// TwinCAT 3 PLC project VLSVacuum
// ProgramVersion: 3.1.4023.0
// libraries:
//   L2SI Vacuum Library, * (SLAC)
//   LCLS General, * (SLAC)
//   LCLSVacuumSerialDriverLib, * (SLAC)
//   PMPS, * (SLAC - LCLS)
//   Tc2_SerialCom, * (Beckhoff Automation GmbH)
//   Tc2_Standard, * (Beckhoff Automation GmbH)
//   Tc2_System, * (Beckhoff Automation GmbH)
//   Tc3_Module, * (Beckhoff Automation GmbH)
// project tree:
//   DUTs/ E_STATES.TcDUT (not stored), ST_VRC_NO.TcDUT
//   GVLs/ GVL_COM_VLS.TcGVL (not stored), GVL_PMPS.TcGVL, GVL_VLS.TcGVL
//   / PlcTask.TcTTO (not stored), VLSSerial.TcTTO
//   POUs/ FB_Pfeffier_NoFault_NO.TcPOU, FB_ValveBase_VLS.TcPOU, FB_VGC_VLS.TcPOU, FB_VRC_NO.TcPOU, FB_VRC_NO_FFO_VLS.TcPOU (not stored), MAIN.TcPOU, PRG_PUMP.TcPOU (not stored), PRG_COM.TcPOU (not stored), PRG_VLS_VACUUM.TcPOU, PRG_VLS_WINDOW.TcPOU
// real-time tasks:
//   TASK PlcTask: cycle T#10ms, priority 20, ADS port 350
//   TASK VLSSerial: cycle T#10ms, priority 1, ADS port 351
// I/O:
//   DEVICE Device 1 (EtherCAT), AmsNetId 172.21.132.45.2.1
//     VLS_Term 1 (EK1200)
//     VLS_EP1 (EP2624-0002)
//     VLS_EP2 (EP2338-0001) [EP2338-0001 8 Ch. Dig. Input/Output 24V, 0,5A, M8]
//     VLS_EP3 (EP2339-0021)
//     VLS_EP4 (EP3174-0002) [EP3174-0002 4Ch. Ana. Input +/-10V, 0-10V, 0/4-20mA configurable]
//     VLS_EP5 (EP6002-0002) [EP6002-0002 Interface (RS232/422/485)]
// variable links:
//   VLSVacuum Instance <-> Device 1 (EtherCAT)/VLS_EP1 (EP2624-0002)
//     PlcTask Outputs/GVL_VLS.DS_GCC.q_xHV_DIS <-> Channel 1/Output
//     PlcTask Outputs/GVL_VLS.PTM_01.q_RunDO <-> Channel 3/Output
//   VLSVacuum Instance <-> Device 1 (EtherCAT)/VLS_EP2 (EP2338-0001)
//     PlcTask Inputs/GVL_VLS.PTM_01.i_xAtSpd <-> Channel 1/Input
//     PlcTask Inputs/GVL_VLS.PTM_01.i_xFaultNC <-> Channel 2/Input
//   VLSVacuum Instance <-> Device 1 (EtherCAT)/VLS_EP3 (EP2339-0021)
//     PlcTask Inputs/GVL_VLS.VGC_1.i_xClsLS <-> Channel 7/Input
//     PlcTask Inputs/GVL_VLS.VGC_1.i_xOpnLS <-> Channel 6/Input
//     PlcTask Inputs/GVL_VLS.VGC_W.i_xClsLS <-> Channel 10/Input
//     PlcTask Inputs/GVL_VLS.VGC_W.i_xOpnLS <-> Channel 9/Input
//     PlcTask Outputs/GVL_VLS.VGC_1.q_xOPN_DO <-> Channel 21/Output
//     PlcTask Outputs/GVL_VLS.VGC_W.q_xCLS_DO <-> Channel 24/Output
//   VLSVacuum Instance <-> Device 1 (EtherCAT)/VLS_EP4 (EP3174-0002)
//     PlcTask Inputs/GVL_VLS.DS_GCC.i_iPRESS_R <-> AI Standard Channel 2/Value
//     PlcTask Inputs/GVL_VLS.DS_GPI.i_iPRESS_R <-> AI Standard Channel 1/Value
//     PlcTask Inputs/GVL_VLS.ROUGH_GPI.i_iPRESS_R <-> AI Standard Channel 3/Value
//   VLSVacuum Instance <-> Device 1 (EtherCAT)/VLS_EP5 (EP6002-0002)
//     VLSSerial Inputs/GVL_COM_VLS.stComIn/D[{0..21}] <-> COM TxPDO-Map Inputs Channel 1/Data In {0..21}  (22 links)
//     VLSSerial Inputs/GVL_COM_VLS.stComIn/Status <-> COM TxPDO-Map Inputs Channel 1/Status
//     VLSSerial Outputs/GVL_COM_VLS.stComOut/Ctrl <-> COM RxPDO-Map Outputs Channel 1/Ctrl
//     VLSSerial Outputs/GVL_COM_VLS.stComOut/D[{0..21}] <-> COM RxPDO-Map Outputs Channel 1/Data Out {0..21}  (22 links)

CONFIGURATION VLSVacuum
    RESOURCE PLC ON TwinCAT3
        TASK VLSSerial(INTERVAL := T#10ms, PRIORITY := 1);
        PROGRAM PRG_COM WITH VLSSerial : PRG_COM;
    END_RESOURCE
END_CONFIGURATION

// ---- DUTs/ST_VRC_NO.TcDUT
TYPE ST_VRC_NO EXTENDS ST_ValveBase:
STRUCT
(* Readbacks *)
	//In case VRC is normally open
	{attribute 'pytmc' := '
    pv: CLS_OK;
	field: ONAM CLOSE; 
	field: ZNAM OPEN;
	io: i;
    '}
	xCLS_OK : BOOL := TRUE;
	{attribute 'pytmc' := '
	pv: CLS_SW ;
	field: ONAM CLOSE; 
	field: ZNAM OPEN;
	io: io ;
	'}
	pv_xCLS_SW	: BOOL;
	{attribute 'pytmc' := '
    pv: FORCE_CLS;
	field: ONAM CLOSE; 
	field: ZNAM OPEN;
	io: io;
	'}
	pv_xOvrdCls	:	BOOL;

END_STRUCT
END_TYPE

// ---- GVLs/GVL_PMPS.TcGVL

VAR_GLOBAL

{attribute 'pytmc' := '
    pv: PLC:TST:FF1
    '}
    {attribute 'TcLinkTo' := '.q_xFastFaultOut:=TIIB[PMPS_FFO]^Channel 1^Output'}
    g_FastFaultOutput1  :   FB_HardwareFFOutput;
	
	{attribute 'pytmc' := '
    pv: PLC:TST:FF2
    '}
    {attribute 'TcLinkTo' := '.q_xFastFaultOut:=TIIB[PMPS_FFO]^Channel 2^Output'}
    g_FastFaultOutput2  :   FB_HardwareFFOutput; 
	fbArbiter: FB_Arbiter(1);
	
END_VAR

// ---- GVLs/GVL_VLS.TcGVL
//{attribute 'qualified_only'}
VAR_GLOBAL

	(* OverrideMode *)
	{attribute 'pytmc' := 'pv: VLS:VAC:OVRDON'}
	xSystemOverrideMode_VLS	: BOOL := FALSE; 	

	(* Pfeiffer Turbo Pumps TM700 *)
	{attribute 'TcLinkTo' := 	'.i_xAtSpd			:=	TIIB[VLS_EP2 (EP2338-0001)]^Channel 1^Input;
								 .i_xFaultNC		:=	TIIB[VLS_EP2 (EP2338-0001)]^Channel 2^Input;
								 .q_RunDO			:=	TIIB[VLS_EP1 (EP2624-0002)]^Channel 3^Output;
			 
	'}
	{attribute 'pytmc' := '
		pv: VLS:PTM:01
		io: io
	'}
    PTM_01 : FB_PTM_Pfeiffer;
	PTM_01_xExtIlkOK : Bool;

	// They share the same serial port
	st_Pfeiffer_CTRL 	: ARRAY[1..20] OF ST_PfeifferControl;
	st_Pfeiffer_RBK 	: ARRAY[1..20] OF ST_PfeifferStatus;
	
	fb_PfeifferCom : FB_PFEIFFER_COM;
	
	
	(* Valves *)
	
	{attribute 'pytmc' :=' pv: VLS:VGC:01 '}
	{attribute 'TcLinkTo' := 	'.i_xOpnLS	:=	TIIB[VLS_EP3 (EP2339-0021)]^Channel 6^Input;
								 .i_xClsLS	:=	TIIB[VLS_EP3 (EP2339-0021)]^Channel 7^Input;
								.q_xOPN_DO	:=	TIIB[VLS_EP3 (EP2339-0021)]^Channel 21^Output'}
	VGC_1 : FB_VGC;
	
	{attribute 'pytmc' :=' pv: VLS:VWC:01 '}
	{attribute 'TcLinkTo' := 	'.i_xOpnLS	:=	TIIB[VLS_EP3 (EP2339-0021)]^Channel 9^Input;
								 .i_xClsLS	:=	TIIB[VLS_EP3 (EP2339-0021)]^Channel 10^Input;
								.q_xCLS_DO	:=	TIIB[VLS_EP3 (EP2339-0021)]^Channel 24^Output'}	
	VGC_W : FB_VRC_NO_FFO_VLS; // Is the Window valve NO 
	
	(* Gauges *)
	
	{attribute 'pytmc' :=' pv: VLS:US:GPI '}
	US_GPI	: FB_MKS275;

	{attribute 'pytmc' :=' pv: VLS:US:GCC '}
	US_GCC	: FB_MKS500;

	{attribute 'pytmc' :=' pv: VLS:DS:GPI '}
	{attribute 'TcLinkTo' := 	'.i_iPRESS_R	:=	TIIB[VLS_EP4 (EP3174-0002)]^AI Standard Channel 1^Value		'}
	DS_GPI	: FB_MKS275;

	{attribute 'pytmc' :=' pv: VLS:DS:GCC '}
	{attribute 'TcLinkTo' := 	'.i_iPRESS_R	:=	TIIB[VLS_EP4 (EP3174-0002)]^AI Standard Channel 2^Value;
								 .q_xHV_DIS		:= 	TIIB[VLS_EP1 (EP2624-0002)]^Channel 1^Output	'}		
	DS_GCC	: FB_MKS500;
	
	{attribute 'pytmc' :=' pv: VLS:ROUGH1:GPI '}
	{attribute 'TcLinkTo' := 	'.i_iPRESS_R	:=	TIIB[VLS_EP4 (EP3174-0002)]^AI Standard Channel 3^Value	'}	
	ROUGH_GPI : FB_9XX;
	
	


END_VAR

// ---- POUs/FB_Pfeffier_NoFault_NO.TcPOU
FUNCTION_BLOCK FB_Pfeffier_NoFault_NO EXTENDS FB_Pump
(* This function block does basic controls FOR the Pfeiffer Turbo pump connected to the TM700 and TC400 Controllers.
 Turns off pump in the event of errors/ warnings. Provides interlocking interface.*)

VAR_IN_OUT
	
END_VAR
VAR_INPUT
	i_xExtIlkOK : BOOL; // Connect to external interlock logic, TRUE if not used.
END_VAR
VAR_OUTPUT
	{attribute 'pytmc' := '
    pv: 
	'}
	iq_stPTM : ST_PfeifferPTM;
END_VAR
VAR
	TOF_RESET: TON :=(PT:=T#1S);
	(*IO*)
	i_xAtSpd AT%I*: BOOL; // Normaml operation when true
	i_xFaultNO AT%I*: BOOL; // Error
	i_xWarn AT%I*: BOOL;
 	i_xRemote AT%I*: BOOL;
	
	q_RunDO AT%Q*: BOOL; // Start/Stop for TC110 link this output to the Pumping station bit
	q_PumpingStation AT%Q*: BOOL; // Start/Stop interlock
	q_xRemote AT%Q*: BOOL;
	q_xReset AT%Q*: BOOL;
END_VAR

(* Basic pump supervisory section *)

q_xRemote := TRUE;
(* Interlock Sum *)
iq_stPtm.xExtRunOk:= i_xExtILKOk;
//For compatability with TC110
(*IF iq_stPTM.xExtRunOk THEN
	q_PumpingStation:= TRUE;
ELSE 
	q_PumpingStation:= FALSE;
END_IF*)

IF iq_stPTM.xExtRunOk AND NOT (iq_stPTM.i_xFault) (*OR iq_stPTM.i_xTempFault)*) THEN
	iq_stPTM.q_RunDO:=iq_stPTM.xRunSW;
	q_PumpingStation:=iq_stPTM.xRunSW;
ELSE
	iq_stPTM.xRunSW:=FALSE;
	iq_stPTM.q_RunDO:=FALSE;
	q_PumpingStation:=FALSE;
	//q_xRemote := TRUE;
END_IF


(*Pump STATE*)
IF iq_stPtm.i_xFault THEN 
	iq_stPtm.eState := pumpFAULT;
ELSIF NOT iq_stPtm.q_RunDO AND NOT iq_stPTM.i_xFault THEN
	iq_stPtm.eState := pumpSTOPPED;
ELSIF NOT iq_stPtm.i_xAtSpd  AND iq_stPtm.q_RunDO THEN
	iq_stPtm.eState := pumpSTARTING;
ELSIF iq_stPtm.i_xAtSpd AND iq_stPtm.q_RunDO THEN
	iq_stPtm.eState := pumpRUNNING;
ELSE 
	iq_stPtm.eState := pumpFAULT;
END_IF

(*Error Reset*)
(* to reset the Reset Bit *)
 IF (iq_stPTM.xResetSW ) THEN  
	iq_stPTM.q_xReset := TRUE; 
	q_PumpingStation := TRUE;
 END_IF

 IF (iq_stPTM.xResetSW) AND (iq_stPTM.i_xFault)  THEN  
	q_PumpingStation := TRUE;
 END_IF
 TOF_RESET (IN:= iq_stPTM.q_xReset, Q => );
 IF TOF_RESET.Q THEN 
	iq_stPTM.q_xReset:= FALSE;
	iq_stPTM.xResetSW := FALSE; 
 END_IF

(*Soft IO Mapping*)
ACT_IO();
// Log States and triggers
ACT_Logger();

ACTION ACT_IO:
(*outputs*)
q_RunDO := iq_stPTM.q_RunDO;
q_xReset := iq_stPTM.q_xReset;
//q_xRemote := iq_stPTM.
//q_PumpingStation AT%Q*: BOOL; // Start/Stop
	
(*inputs*)
iq_stPTM.i_xAtSpd:= i_xAtSpd;
iq_stPTM.i_xFault:= i_xFaultNO; 
iq_stPTM.i_xWarn:=  	i_xWarn ;
END_ACTION

ACTION ACT_Logger:
//STATE Logger  
IF NOT i_xExtIlkOK AND ePrevState = pumpRUNNING THEN
 		fbLogger(sMsg:='Lost external interlock while pump was running.', eSevr:=TcEventSeverity.Critical);  	
END_IF


IF ePrevState <> iq_stPTM.eState THEN
	  CASE iq_stPTM.eState OF
		pumpFAULT:
			fbLogger(sMsg:='Pump Fault.', eSevr:=TcEventSeverity.Critical);
  		pumpSTOPPED:
			fbLogger(sMsg:='Pump stopped.', eSevr:=TcEventSeverity.Critical);
		pumpSTARTING:
			fbLogger(sMsg:='Pump starting.', eSevr:=TcEventSeverity.Info);
		pumpRUNNING:
			fbLogger(sMsg:='Pump running.', eSevr:=TcEventSeverity.Info);
	  END_CASE
	  ePrevState := iq_stPTM.eState;  
  END_IF
  
// ILK logger



// Log Action
tAction(CLK:=  iq_stPTM.q_RunDO);
IF tAction.Q THEN fbLogger(sMsg:='Pump commanded to start', eSevr:=TcEventSeverity.Info); END_IF


// Log FAULT
tFault(CLK:= NOT iq_stPTM.i_xFault);
IF tFault.Q THEN fbLogger(sMsg:='Pump Lost Alarm OK bit', eSevr:=TcEventSeverity.Critical); END_IF
END_ACTION

METHOD PUBLIC M_Serial_IO : BOOL
VAR_INPUT
	st_Pfeiffer_RBK: ST_PfeifferStatus;
END_VAR
VAR_IN_OUT
	st_Pfeiffer_CTRL: ST_PfeifferControl;
END_VAR
(* This function block is used to map the IO points from the pfeiffer structures
to the generic turbo structures *)
(*
if (bInit) Then
	bInit := False;
	st_Pfeiffer_CTRL.diSetRotationSpeed_309 := st_Pfeiffer_RBK.diActiveRotationSpeed_309;
END_IF*)

(* Controls *) (* Controls is via DIO*)
st_Pfeiffer_CTRL.xPumpingStation_010 := iq_stPTM.q_RunDO;
//st_Pfeiffer_CTRL.xMotorPump_023 := 1; //Setting always true because parameter 10 alone can enable/disable the pump
//st_Pfeiffer_CTRL.uiPowerPct_708 := iq_stPTM.q_uiPowerPct;
//st_Pfeiffer_CTRL.xErrorAck_009 := iq_stPTM.xResetSW;



(* Readbacks *)
iq_stPTM.i_xAccel := st_Pfeiffer_RBK.xPumpAccelerating_307;
//iq_stPTM.i_xAtSpd := st_Pfeiffer_RBK.xRotationSpeedAttn_306; The Atspd is already linked via Digital I/Os
iq_stPTM.i_diCurSpd := st_Pfeiffer_RBK.diActiveRotationSpeed_309;
iq_stPTM.i_diPwr := st_Pfeiffer_RBK.diDrivePower_316;
iq_stPTM.i_diElecTemp := st_Pfeiffer_RBK.diTempElec_326;
iq_stPTM.i_diBtmTemp := st_Pfeiffer_RBK.diTempPmpBot_330;
iq_stPTM.i_diBrngTemp := st_Pfeiffer_RBK.diTempBearng_342;
iq_stPTM.i_diMtrTemp := st_Pfeiffer_RBK.diTempMotor_346;
iq_stPTM.i_uiPowerPctRbk := st_Pfeiffer_RBK.uiPowerPct_708;
iq_stPTM.i_rCurrentMon :=  st_Pfeiffer_RBK.lrDriveCurrent_310;
iq_stPTM.xCommTimeout	:=	st_Pfeiffer_RBK.xTimeout;
iq_stPTM.i_iErrorCode := st_Pfeiffer_RBK.iErrorCode_303;
iq_stPTM.i_iWarningCode := st_Pfeiffer_RBK.iWarningCode_303;

(* Check that error acknowledgment is processed *)
IF st_Pfeiffer_RBK.xErrorAcknowledged THEN
	st_Pfeiffer_RBK.xErrorAcknowledged := FALSE;
	st_Pfeiffer_CTRL.xErrorAck_009 := FALSE;
	iq_stPTM.xResetSW := FALSE;
END_IF

IF st_Pfeiffer_RBK.sErrorCode_303 = '' THEN
	;
ELSIF st_Pfeiffer_RBK.sErrorCode_303 <> '000000' THEN
iq_stPTM.i_xFault := TRUE;
ELSE
iq_stPTM.i_xFault := FALSE;
END_IF

iq_stPTM.i_dSetSpd := LIMIT (0, iq_stPTM.i_dSetSpd, 1500); // 1500 nominal frequency
IF ( iq_stPTM.i_dSetSpd <>0) THEN
	st_Pfeiffer_CTRL.iSetRotationSpeed_707 := DINT_TO_INT(iq_stPTM.i_dSetSpd * 100/1500);
	st_Pfeiffer_CTRL.iSetRotationSpeed_707 := LIMIT(20, st_Pfeiffer_CTRL.iSetRotationSpeed_707 ,100); // Manual Page 18
END_IF
END_METHOD

END_FUNCTION_BLOCK

// ---- POUs/FB_ValveBase_VLS.TcPOU
FUNCTION_BLOCK FB_ValveBase_VLS
VAR_INPUT
END_VAR
VAR_OUTPUT
END_VAR
VAR
	// For logging
    fbLogger : FB_LogMessage := (eSubsystem:=E_SubSystem.VACUUM);
   // ePrevState : E_ValvePositionState;
    tErrorPresent : R_TRIG;
    tAction : R_TRIG; // Primary action of this device (OPN_DO, etc.)
    tOverrideActivated : R_TRIG;
END_VAR

ACTION ACT_Logger:

END_ACTION

END_FUNCTION_BLOCK

// ---- POUs/FB_VGC_VLS.TcPOU
(* This function block implements basic functionality for Isolation Gate Valves*)
(* This function block interlock is as follows:
1. The valve can be opened when the difference between the pressures on both sides is
less than the maximum differential pressure.
2. This rule persists until the pressures on both sides are lower than the vacuum-setpoint.
3. Once at-vac, the valve will close if the pressure on either side rises above the setpoint.*)
(*This function block also implements PMPS and EPS interlocks, as well as Fast MPS trigger*)
FUNCTION_BLOCK FB_VGC_VLS Extends FB_ValveBase
VAR_IN_OUT
END_VAR
VAR_INPUT
	(*Upstream Gauge, usually ion gauge*)
	i_stUSG	:	ST_VG;
	(*Downstream Gauge, usually ion gauge*)
	i_stDSG	:	ST_VG;
	{attribute 'pytmc' := '
    pv: Dis_DPIlk
	'}
	i_xDis_DPIlk : BOOL := FALSE;  (* Set to true when calling the function to disable the differential pressure interlock *)
	{attribute 'pytmc' := '
    pv: EPS_OPN_OK
	'}
	i_xEPS_OPN_OK:	BOOL	:= TRUE; (*External EPS interlock, Set to TRUE when no EPS interlock is required, otherwise set to correct interlock signal*)
	{attribute 'pytmc' := '
    pv: EPS_CLS_OK
	'}
	i_xEPS_CLS_OK:	BOOL	:= TRUE; (*External EPS interlock, Set to TRUE when no EPS interlock is required, otherwise set to correct interlock signal*)
	
	{attribute 'pytmc' := '
    pv: MPS_OK
	'}
	i_xPMPS_OK:	BOOL	; (*External MPS interlock, Set to TRUE when no PMPS interlock is required*)
	i_xExt_OK: BOOL; (*Other External Interlock, Set to True when no external interlock is required. If this Valve is neigboring a Fast Shutter this should be linked to the fast shutter xVAC_FAULT_OK*)
	i_xOverrideMode : BOOL; (*To be linked to global override bit. This Overrides Vacuum logic only, EPS, MPS and PMPS are still enforces*)
	// Reset fault
	{attribute 'pytmc' := '
    pv: FF_Reset
	'}
    i_xReset: BOOL;
END_VAR
VAR_OUTPUT
	{attribute 'pytmc' := '
    pv:
	'}
	iq_stValve : ST_VGC; (* All valve data and states will be in this struct*)
	
END_VAR

VAR
	{attribute 'instance-path'}
	{attribute 'noinit'}
	sPath: STRING;
	rDiffPressAllowed	:	REAL := 22.5; // Torr, Default value comes from Vat Valve Manual
	rDiffPress : REAL;
	set : BOOL;
    reset: BOOL;
	  
	xFirstPass	:	BOOL;
	fbFSInit		:	R_TRIG;
	
	tonDelOK : TON;
	rtOK	:	R_TRIG;
	tonOvrd	:	TON;
	rtOpen	:	R_TRIG;
	ftClose: F_TRIG;
	
	tDelOK	:	TIME := T#60S;
	tOvrd	:	TIME := T#10s;
	ePrevState : E_VGC;
	
	(* Timeouts*)
	tTimeOutDuration: TIME:= T#10S;
	tOPNtimeout: TON;
	tCLStimeout:TON;
	
	
	
	(*IO*)
	i_xOpnLS	AT%I*: BOOL;
	i_xClsLS	AT%I*: BOOL;
	q_xOPN_DO	AT%Q*: BOOL;
    
  
END_VAR

(* Vacuum gate valve
A. Wallace
16-10-29

A gate valve isolates vacuum volumes. Ideally it can be opened when a system is vented
to allow for faster pumping, and will close when high vacuum is lost.

The following behavior is good for valves in something like a gas attenuator.
This function block does the following:
1. The valve can be opened when the difference between the pressures on both sides is
less than the maximum differential pressure.
2. This rule persists until the pressures on both sides are lower than the vacuum-setpoint.
3. Once at-vac, the valve will close if the pressure on either side rises above the setpoint.

Alternatively, the differential pressure interlock can be disabled so the valve may only be opened
if the pressure on both sides is lower than the at-vacuum-setpoint. You want this behavior if 
the valve is to be used in a UHV section.

Hysteresis is employed to ensure a smooth transition from vented/pumping down, to at-vac.

Finally, an override system is built in so you can bypass all the interlocking logic and 
get back online.
*)
(* 10/1/2018 Margaret Ghaly included EPS, PMPS Checkes and MPS trigger signals*)

ACT_Init();
(*IO Mapping*)
ACT_IO();
A_Override();
A_PositionCheck();
ACT_ResetAlarms();
A_EPS();
// Main logic the very last call right before IO
ACT_Main();
(*IO Mapping*)
ACT_IO();
A_Logger();

ACTION A_EPS:
ftClose(CLK:= iq_stValve.pv_xOPN_SW);
rtOpen(CLK:= iq_stValve.pv_xOPN_SW);


(* If Epics Command to close the Valve, check if PMPS and EPS are ok, otherwise Keep command set to open valve *)
// Check a falling edge on the open switch, which means that the valve is commanded to close
IF (ftClose.Q) THEN
	// check that the valve is allowed to close, and that it was already in the open position otherwise, he command is to be ingonred and reset
	IF NOT(i_xEPS_CLS_OK) AND (iq_stValve.q_xOPN_DO) THEN iq_stValve.pv_xOPN_SW := TRUE; END_IF;
END_IF

// if switch pv has been switched to open
IF (rtOpen.Q) THEN 
	// if the EPS interlock the valve from openening, the switch pv is reset to false i.e ignoring the action
	IF NOT (i_xEPS_OPN_OK) THEN  iq_stValve.pv_xOPN_SW := FALSE; END_IF
END_IF
END_ACTION

ACTION A_Logger:
// Log valve timeouts
tErrorPresent(CLK:=iq_stValve.bErrorPresent);
IF tErrorPresent.Q THEN fbLogger(sMsg:=iq_stValve.sErrorMessage, eSevr:=TcEventSeverity.Warning); END_IF

// Log valve open
tAction(CLK:= iq_stValve.q_xOPN_DO);
IF tAction.Q THEN fbLogger(sMsg:='Valve commanded open', eSevr:=TcEventSeverity.Info); END_IF

// Log override mode enabled
tOverrideActivated(CLK:= (tonOvrd.Q AND i_xOverrideMode));
IF tOverrideActivated.Q THEN fbLogger(sMsg:='Valve override mode activated', eSevr:=TcEventSeverity.Warning); END_IF
END_ACTION

ACTION A_Override:
(* Override logic *)
(* Goal: give ability to override, but do so in a way that people won't forget it.
Solution: Override only after ten seconds of override, protect against blips,
when the valve permission goes true for more than ten seconds consistently, remove override
*)

tonDelOK(IN:=iq_stValve.xOPN_OK, PT:=tDelOK);
rtOK(CLK:=tonDelOK.Q);
IF rtOK.Q AND iq_stValve.pv_xOvrdOpn THEN 
	if (iq_stValve.eState = OPEN) AND (i_xOverrideMode) AND (iq_stValve.pv_xOvrdOpn) THEN iq_stValve.pv_xOPN_SW := TRUE; END_IF //for seamless transition   
   	iq_stValve.pv_xOvrdOpn :=FALSE; // reset the overrride open bit
	//Log
    fbLogger(sMsg:='Override expired', eSevr:=TcEventSeverity.Warning);
    
END_IF

//Override timer
tonOvrd(IN:=iq_stValve.pv_xOvrdOpn, PT:=tOvrd);
END_ACTION

ACTION A_PositionCheck:


///Check valve position
IF iq_stValve.i_xClsLS AND  iq_stValve.i_xOpnLS THEN
	iq_stValve.eState:=INVALID;
ELSIF NOT iq_stValve.i_xClsLS AND iq_stValve.i_xOpnLS AND iq_stValve.q_xOPN_DO THEN 
	iq_stValve.eState:=OPEN;
ELSIF iq_stValve.i_xClsLS AND NOT iq_stValve.i_xOpnLS AND NOT iq_stValve.q_xOPN_DO THEN 
	iq_stValve.eState:=CLOSED;
ELSIF NOT iq_stValve.i_xClsLS AND NOT iq_stValve.i_xOpnLS THEN 
	iq_stValve.eState:=MOVING;
ELSE
	iq_stValve.eState:=INVALID;
END_IF


///Check valve moving postion timout
IF NOT iq_stValve.i_xClsLS AND tCLStimeout.Q THEN 
	iq_stValve.bErrorPresent := TRUE;
	iq_stValve.sErrorMessage := ' Close Timeout';
ELSIF NOT iq_stValve.i_xOpnLS AND tOPNtimeout.Q THEN 
	iq_stValve.bErrorPresent := TRUE; 
	iq_stValve.sErrorMessage := ' Open Timeout';
END_IF
IF (iq_stValve.eState=INVALID) THEN
	iq_stValve.bErrorPresent := TRUE; 
	iq_stValve.sErrorMessage := CONCAT(sPath,' Invalid Valve Position');
END_IF


(*Timers*)
tOPNtimeout(IN:= iq_stValve.q_xOPN_DO, PT := tTimeOutDuration );
tCLStimeout(IN:= NOT iq_stValve.q_xOPN_DO, PT := tTimeOutDuration);
END_ACTION

ACTION ACT_Init:
fbFSInit( CLK := TRUE, Q => xFirstPass);
(* On first PLC pass, put valve into vented state, which implies a closed valve *)
IF xFirstPass THEN
	iq_stValve.eVGC_State := Vented;
	iq_stValve.pv_xOPN_SW := FALSE;
END_IF
END_ACTION

ACTION ACT_IO:
(*inputs*)
iq_stValve.i_xOpnLS := 	i_xOpnLS;
iq_stValve.i_xClsLS:=	i_xClsLS;
iq_stValve.xEXT_OK := i_xEXT_OK;
iq_stValve.xOverrideMode := i_xOverrideMode;
(*outputs*)
q_xOPN_DO:= iq_stValve.q_xOPN_DO;
END_ACTION

ACTION ACT_Main:

// Update hysteresis
///////////////////////////////////////////////////
IF iq_stValve.rAT_VAC_SP_LAST <> iq_stValve.rAT_VAC_SP OR xFirstPass THEN
	iq_stValve.rAT_VAC_SP_LAST := iq_stValve.rAT_VAC_SP;
	iq_stValve.rAT_VAC_HYS := iq_stValve.rHYST_PERC * iq_stValve.rAT_VAC_SP;
END_IF

iq_stValve.rAT_VAC_HYS := LIMIT(0, iq_stValve.rAT_VAC_HYS, iq_stValve.rAT_VAC_SP);
IF iq_stValve.rAT_VAC_SP <> 0 THEN
	IF iq_stValve.rHYST_PERC <> (iq_stValve.rAT_VAC_HYS / iq_stValve.rAT_VAC_SP) THEN
		iq_stValve.rHYST_PERC := LIMIT(0, (iq_stValve.rAT_VAC_HYS / iq_stValve.rAT_VAC_SP) ,1);
	END_IF
END_IF
// Valve at vacuum check
///////////////////////////////////////////////////
	set := i_stUSG.rPRESS < iq_stValve.rAT_VAC_HYS AND i_stDSG.rPRESS < iq_stValve.rAT_VAC_HYS AND i_stUSG.xPRESS_OK AND i_stDSG.xPRESS_OK;
 	iq_stValve.xAT_VAC S= set;
	reset := i_stUSG.rPRESS > iq_stValve.rAT_VAC_SP OR i_stDSG.rPRESS > iq_stValve.rAT_VAC_SP OR NOT i_stUSG.xPRESS_OK OR NOT i_stDSG.xPRESS_OK;
	iq_stValve.xAT_VAC R= reset;
	
// Differential pressure check
///////////////////////////////////////////////////
	(* Calc the differential pressure across the valve *)
	rDiffPress := ABS(i_stUSG.rPRESS - i_stDSG.rPRESS);
	
	(* As long as the differential pressure is less than 30mbar, the valve is allowed to open *)
	IF rDiffPress <= rDiffPressAllowed AND i_stUSG.xPRESS_OK AND i_stDSG.xPRESS_OK THEN
		iq_stValve.xDP_OK := TRUE;
	ELSE
		iq_stValve.xDP_OK	:= FALSE;
		(* If the differential pressure is exceeded, even when the valve is open,
		the state is unexpected and triggers a fault, because it suggests that something
		is wrong with the valve, or gauges or mapping or there is a major leak on one side.*)
		iq_stValve.eVGC_State := ERR_DiffPress;
        iq_stValve.xERR_DifPres := TRUE;
	END_IF

// Valve state
///////////////////////////////////////////////////
CASE iq_stValve.eVGC_State OF
	Vented: (* The Vented state is used during pump down *)
        //Log new state
        IF ePrevState <> iq_stValve.eVGC_State THEN
            fbLogger(sMsg:='Vented', eSevr:=TcEventSeverity.Info);
            ePrevState := iq_stValve.eVGC_State;
		END_IF
        
		(* Assuming the pump down went well, we are now at vacuum on both sides,
		so we move to the vacuum state, otherwise remain in the vented state *)
		IF iq_stValve.xAT_VAC AND (NOT (iq_stValve.xERR_DifPres)) AND NOT (NOT (iq_stValve.xERR_SP)) and NOT (NOT (iq_stValve.xERR_ExtFault))THEN
		    iq_stValve.eVGC_State := AtVacuum;
		ELSE
		    iq_stValve.eVGC_State := Vented;
		END_IF
	
	AtVacuum:
        //Log new state
        IF ePrevState <> iq_stValve.eVGC_State THEN
            fbLogger(sMsg:='Vacuum setpoint satisfied', eSevr:=TcEventSeverity.Info);
            ePrevState := iq_stValve.eVGC_State;
		END_IF
        
		IF iq_stValve.xAT_VAC THEN
		(* If both pressure setpoints are made,
		then enable the differential pressure interlock, regardless of the valve state
		assuming we're using some kind of ion gauge where a pressure setpoint cannot be higher than 1E-4 T *)
		iq_stValve.eVGC_State := AtVacuum;
				
		ELSE
		
			(* If the valve is open (or in an unknown state) and either gauge is not at it's vacuum setpoint,
			we have a loss of vacuum error *)
			IF (iq_stValve.i_xOpnLS OR (NOT iq_stValve.i_xOpnLS AND NOT iq_stValve.i_xClsLS)) THEN
				iq_stValve.eVGC_State := ERR_LostVac;
				iq_stValve.xERR_SP := TRUE; //TAW changed this to the ERR_SP bool because I think that's what it was intended to be?
		
			(* Alternatively, if the valve is already closed and we lose pressure on one side,
			it was probably intentional venting, so we calmly move back to venting mode, and
			disable the differential pressure interlock *) //?? 
			ELSIF iq_stValve.i_xClsLS THEN
				iq_stValve.eVGC_State := Vented;
			END_IF
		
		END_IF
	
	ERR_DiffPress:
        //Log new state
        IF ePrevState <> iq_stValve.eVGC_State THEN
            fbLogger(sMsg:='Potential accidental vent.', eSevr:=TcEventSeverity.Critical);
            ePrevState := iq_stValve.eVGC_State;
		END_IF
        
		IF NOT (iq_stValve.xERR_DifPres) THEN
			iq_stValve.eVGC_State := Vented;
		END_IF
		
	
	ERR_LostVac:
        //Log new state
        IF ePrevState <> iq_stValve.eVGC_State THEN
            fbLogger(sMsg:='Unexpected loss of vacuum while valve was open.', eSevr:=TcEventSeverity.Critical);
            ePrevState := iq_stValve.eVGC_State;
		END_IF
		IF NOT (iq_stValve.xERR_SP) THEN
			iq_stValve.eVGC_State := Vented;
		END_IF
		
	ERR_ExtFault:
        //Log new state
        IF ePrevState <> iq_stValve.eVGC_State THEN
            fbLogger(sMsg:='Lost external interlock while valve was open.', eSevr:=TcEventSeverity.Critical);
            ePrevState := iq_stValve.eVGC_State;
		END_IF
		IF NOT (iq_stValve.xERR_ExtFault) AND (NOT i_xExt_OK) THEN
			iq_stValve.eVGC_State := Vented;
		END_IF
END_CASE

IF (NOT i_xExt_OK) THEN
	iq_stValve.eVGC_State := ERR_ExtFault;
	iq_stValve.xERR_ExtFault := TRUE;
END_IF

// Interlock evaluation - with bypass for DP ILK bypass
///////////////////////////////////////////////
IF i_xDis_DPIlk THEN
	iq_stValve.xOPN_OK := iq_stValve.xEXT_OK; // AND iq_stValve.xDP_OK ;
ELSE
	iq_stValve.xOPN_OK := iq_stValve.xEXT_OK AND iq_stValve.xAT_VAC;
END_IF

(* Valve operation *)
if NOT (iq_stValve.xOPN_OK) THEN iq_stValve.pv_xOPN_SW:= FALSE; END_IF // redundant??
(* Here's where the valve opens *)
iq_stValve.q_xOPN_DO := (iq_stValve.pv_xOPN_SW AND iq_stValve.xOPN_OK) OR (tonOvrd.Q AND i_xOverrideMode);
END_ACTION

ACTION ACT_ResetAlarms:
iq_stValve.xERR_DifPres R= iq_stValve.pv_xAlmRst;
iq_stValve.xERR_SP R= iq_stValve.pv_xAlmRst;
iq_stValve.bErrorPresent R= iq_stValve.pv_xAlmRst;

IF ( iq_stValve.pv_xAlmRst) THEN
	iq_stValve.sErrorMessage :='';
END_IF
END_ACTION

METHOD PUBLIC M_IsClosed : BOOL
VAR_INPUT
END_VAR
M_IsClosed := (This^.iq_stValve.eState = E_ValvePositionState.CLOSED);
END_METHOD

METHOD PUBLIC M_IsOpen : BOOL
VAR_INPUT
END_VAR
M_IsOpen := (This^.iq_stValve.eState = E_ValvePositionState.OPEN);
END_METHOD

// Use this Methode to Open or close the valve by setting the OPN_SW to the input value.
METHOD PUBLIC M_Set_OPN_SW : BOOL
VAR_INPUT
		value:BOOL;
END_VAR
This^.iq_stValve.pv_xOPN_SW := value;
END_METHOD

END_FUNCTION_BLOCK

// ---- POUs/FB_VRC_NO.TcPOU
(* This function block is different from the regular VRC in that CLOSING must be permitted. *)
FUNCTION_BLOCK FB_VRC_NO EXTENDS FB_Valve
VAR_IN_OUT

END_VAR
VAR_INPUT

	i_xExtILK_OK : BOOL; //Connect to Interlock logic condition(e.g F_TURBO_VRC_ILK Function), otherwise, Set to True if the valve is not interlocked
	i_xOverrideMode : BOOL; (*To be linked to global override bit. This Overrides Vacuum logic only, EPS, MPS and PMPS are still enforces*)

END_VAR
VAR_OUTPUT
	{attribute 'pytmc' := '
    pv:
	'}
		iq_stValve : ST_VRC_NO;
END_VAR
VAR

	{attribute 'noinit'}
	sPath: STRING;
	xFirstPass	:	BOOL;
	fbFSInit		:	R_TRIG;
	tonOvrd	:	TON;
	tonDelOK : TON;
	rtOK	:	R_TRIG;
	tOvrd	:	TIME := T#10s;
	(* Timeouts*)
	tTimeOutDuration: TIME:= T#30S;
	tOPNtimeout: TON;
	tCLStimeout:TON;
	

(*IO*)
	i_xOpnLS	AT%I*: BOOL;
	i_xClsLS	AT%I*: BOOL;
	q_xCLS_DO	AT%Q*: BOOL;

END_VAR

(* This function block is different from the regular VRC in that CLOSING must be permitted. *)

(* On first PLC pass, put valve into vented state, which implies a closed valve *)
fbFSInit( CLK := TRUE, Q => xFirstPass);
IF xFirstPass THEN
	iq_stValve.pv_xCLS_SW := FALSE;
END_IF




///Check valve position
IF iq_stValve.i_xClsLS AND  iq_stValve.i_xOpnLS THEN
	iq_stValve.eState:=INVALID;
ELSIF NOT iq_stValve.i_xClsLS AND iq_stValve.i_xOpnLS AND iq_stValve.q_xOPN_DO THEN 
	iq_stValve.eState:=OPEN;
ELSIF iq_stValve.i_xClsLS AND NOT iq_stValve.i_xOpnLS AND NOT iq_stValve.q_xOPN_DO THEN 
	iq_stValve.eState:=CLOSED;
ELSIF NOT iq_stValve.i_xClsLS AND NOT iq_stValve.i_xOpnLS THEN 
	iq_stValve.eState:=MOVING;
ELSE
	iq_stValve.eState:=INVALID;
END_IF


(*evaluate Valve CLose external interlock*)
iq_stValve.xCLS_OK := i_xExtILK_OK;
IF NOT iq_stValve.xCLS_OK and NOT tonOvrd.Q THEN
	iq_stValve.pv_xCLS_SW := FALSE;
END_IF


(* Override logic *)
(* Goal: give ability to override, but do so in a way that people won't forget it.
Solution: Override only after ten seconds of override, protect against blips,
when the valve permission goes true for more than ten seconds consistently, remove override
*)

tonDelOK(IN:=iq_stValve.xCLS_OK, PT:=T#10S);
rtOK(CLK:=tonDelOK.Q);
IF rtOK.Q AND iq_stValve.pv_xOvrdCls THEN 
	iq_stValve.pv_xOvrdCls :=FALSE; 
	if (iq_stValve.eState=CLOSED) AND (i_xOverrideMode) THEN iq_stValve.pv_xCLS_SW := TRUE; END_IF
    //Log
    fbLogger(sMsg:='Override expired', eSevr:=TcEventSeverity.Warning);
END_IF

//Override timer
tonOvrd(IN:=iq_stValve.pv_xOvrdCls, PT:=tOvrd);

(* Here's where the valve Actuates *)
q_xCLS_DO := ((iq_stValve.xCLS_OK  AND iq_stValve.pv_xCLS_SW)OR (tonOvrd.Q AND i_xOverrideMode));
iq_stValve.q_xOPN_DO := NOT q_xCLS_DO;



///Check valve moving position timout
IF NOT iq_stValve.i_xClsLS AND tCLStimeout.Q THEN 
	iq_stValve.bErrorPresent := TRUE;
	//iq_stValve.sErrorMessage := ' Close Timeout';
ELSIF NOT iq_stValve.i_xOpnLS AND tOPNtimeout.Q THEN 
	iq_stValve.bErrorPresent := TRUE; 
	//iq_stValve.sErrorMessage := ' Open Timeout';
END_IF
IF (iq_stValve.eState=INVALID) THEN
	iq_stValve.bErrorPresent := TRUE; 
	//iq_stValve.sErrorMessage := CONCAT(sPath,' Invalid Valve Position');
END_IF

(*Timers*)
tOPNtimeout(IN:= iq_stValve.q_xOPN_DO, PT := tTimeOutDuration );
tCLStimeout(IN:= NOT iq_stValve.q_xOPN_DO, PT := tTimeOutDuration);


(*Soft IO Mapping*)
ACT_IO();

// Log States and triggers
ACT_Logger();

ACTION ACT_IO:
(*inputs*)
iq_stValve.i_xOpnLS := 	i_xOpnLS;
iq_stValve.i_xClsLS:=	i_xClsLS;
//iq_stValve. := i_xEXT_OK;
iq_stValve.xOverrideMode := i_xOverrideMode;
(*outputs*)
//q_xOPN_DO:= iq_stValve.q_xOPN_DO;
END_ACTION

METHOD M_IsClosed : BOOL
VAR_INPUT
END_VAR
M_IsClosed := (This^.iq_stValve.eState = E_ValvePositionState.CLOSED);
END_METHOD

METHOD M_IsOpen : BOOL
VAR_INPUT
END_VAR
M_IsOpen := (This^.iq_stValve.eState = E_ValvePositionState.OPEN);
END_METHOD

METHOD M_Set_CLS_W : BOOL
VAR_INPUT
	value:BOOL;
END_VAR
This^.iq_stValve.pv_xCLS_SW := value;
END_METHOD

END_FUNCTION_BLOCK

// ---- POUs/MAIN.TcPOU
PROGRAM MAIN
VAR
	// Variable for VLS upstream pressure bit
	{attribute 'pytmc' := '
	pv: EXT_PRESS_OK ;
	field: ZNAM NOT OK ;
	field: ONAM OK ;
	io: i ;
	'}
	bVLS_Press_OK : BOOL := FALSE; // TRUE : OK to open gate valve, FALSE : not OK to open gate valve
	
//	stPTM : ST_PfeifferControl;
//	fbPTM : FB_PTM_Pfeiffer;
END_VAR

(* Example main program to show how to incorporate the VLS vacuum program *)

PRG_VLS_VACUUM();

END_PROGRAM

// ---- POUs/PRG_VLS_VACUUM.TcPOU
PROGRAM PRG_VLS_VACUUM
VAR


END_VAR
VAR_INPUT
	bVLS_Ext_Press : BOOL := FALSE; // external interlock bit for window control
END_VAR

// VLS Vacuum Logic
PRG_VLS_WINDOW(bExtPress := bVLS_Ext_Press); // run the vacuum program with interlock bit

// VLS Pump
PRG_PUMP();

END_PROGRAM

// ---- POUs/PRG_VLS_WINDOW.TcPOU
PROGRAM PRG_VLS_WINDOW
VAR
	xFirstPass		: BOOL;
	fbFSInit		: R_TRIG;
	
	state			: E_STATES;

	bOverride		: BOOL;
	bSetup			: BOOL;
	

END_VAR
VAR_INPUT
	bExtPress		: BOOL := FALSE; // Input for external interlock with hutch vacuum system
END_VAR

fbFSInit( CLK := TRUE, Q => xFirstPass);
(* On first PLC pass, put valve into init state*)
IF xFirstPass THEN
	state:= E_STATES.INIT;
	bOverride := FALSE;
	bSetup := FALSE;
END_IF


//STATE ACTIONS
CASE state OF

 E_STATES.INIT: 
		VGC_1.M_Set_OPN_SW(FALSE); //Isolation Valve closed
		VGC_W.M_Set_CLS_SW(FALSE); // Window valve OPEN
		VGC_1.i_xOverrideMode := VGC_W.i_xOverrideMode := FALSE;
		//Transition
		if (VGC_1.M_IsClosed() AND VGC_W.M_IsOpen()) THEN
			state:= E_STATES.NOT_SAFE;
		END_IF
		
E_STATES.NOT_SAFE: // System is not allowed to actuate, i.e all interlocks are in effect
	VGC_1.M_Set_OPN_SW(VGC_1.iq_stValve.q_xOPN_DO );
 	//C_1.i_xExt_OK := VGC_1.i_xEPS_OPN_OK := VGC_1.i_xEPS_CLS_OK:= FALSE; 
	VGC_W.i_xExtILK_OK:= FALSE; 
	VGC_1.i_xOverrideMode := VGC_W.i_xOverrideMode := FALSE;

	//Transition
	//IF (US_GCC.IG.xAT_VAC AND DS_GCC.IG.xAT_VAC) THEN state:= E_STATES.READY; END_IF
	IF (bExtPress AND DS_GCC.IG.xAT_VAC) THEN state:= E_STATES.READY; END_IF
	
	
	
 E_STATES.READY: // OK to MOVE
 	// Release the external interlock so the differential pressure inlk is in effect
 	VGC_1.i_xExt_OK:= VGC_1.i_xEPS_OK :=TRUE;
	//permission to insert window valve only when US vacuum is good??
	VGC_W.i_xExtILK_OK:= bExtPress;
	// Valves  alternate positions.
	If (VGC_W.M_IsClosed()) THEN  VGC_1.M_Set_OPN_SW(TRUE);
	ELSIF (VGC_W.M_IsOpen()) THEN VGC_1.M_Set_OPN_SW(FALSE);
	END_IF
	
 
 E_STATES.OVERRIDE: 
	// Override Mode is enabled for all valves
 	VGC_1.i_xOverrideMode :=VGC_W.i_xOverrideMode := TRUE;
	// Exit of Override mode always goes back to init
 	IF NOT(bOverride) THEN state:= E_STATES.INIT; END_IF
	
	
 E_STATES.SETUP: 
	// Window valve remains retracted
 	VGC_W.i_xExtILK_OK := FALSE; 
	// Isolation valves operates like standard gate valves 
	VGC_1.i_xExt_OK := TRUE;
	// exit to init just to be safe?
	IF NOT(bSetup) THEN state:= E_STATES.INIT; END_IF
END_CASE


// STATE TRANSITIONS
// the system can go to setup state from any other state except override
IF (bSetup) AND (state<>E_STATES.OVERRIDE) THEN state:= E_STATES.SETUP; 
// the system can go to override state from any other state except setup
ELSIF (bOverride) AND (state<>E_STATES.SETUP) THEN state:= E_STATES.OVERRIDE;
//Loss of at vac signal makes the system go to init/not safe to move state
ELSIF (NOT bExtPress) OR (NOT DS_GCC.IG.xAT_VAC) THEN state:= E_STATES.INIT;
//ELSIF (NOT US_GCC.IG.xAT_VAC) OR (NOT DS_GCC.IG.xAT_VAC) THEN state:= E_STATES.INIT;
END_IF 


// Instantiate function blocks
US_GPI(PG=>);
//US_GCC(PG:=US_GPI.PG);
DS_GPI(PG=>);
DS_GCC(PG:=DS_GPI.PG , IG=> , bEP := TRUE );

ROUGH_GPI.M_SetBits(32767);
ROUGH_GPI(PG=>);

VGC_1(
	i_stUSG:= US_GCC.IG , 
	i_stDSG:= DS_GCC.IG , 
	i_xDis_DPIlk:= FALSE , 
	i_xPMPS_OK:= , 
	i_xEPS_OK:= , 
	i_xExt_OK:= , 
	i_xOverrideMode:= , 
	i_xReset:= , 
	i_xIsAperture:= FALSE, 
	i_sDevName:= , 
	i_nTransitionRootID:=  1000,
	iq_stValve=> , 
	xMPS_OK=> , 
	io_fbFFHWO:=g_FastFaultOutput2 , 
	fbArbiter:=fbArbiter);


VGC_W(
	i_xExtILK_OK:= , 
	i_xOverrideMode:= , 
	iq_stValve=> , 
	io_fbFFHWO:= g_FastFaultOutput2 , 
	fbArbiter:= fbArbiter, 
	i_xPMPS_OK:= , 
	i_xIsAperture:= TRUE , 
	i_sDevName:= , 
	i_nTransitionRootID:= 2000);
	
	
//VGC_W(i_xExtILK_OK:= , 
//	i_xOverrideMode:= ,
 //   iq_stValve=> );

END_PROGRAM
